// TIA Portal V18 export
DATA_BLOCK "Debug"   // DB5
{ S7_Optimized_Access := 'TRUE' }
VERSION : 0.1
// stored: AutoNumber false, DBAccessibleFromOPCUA true, DBAccessibleFromWebserver true, IsOnlyStoredInLoadMemory false, IsRetainMemResEnabled false, IsWriteProtectedInAS false, MemoryReserve 100
   VAR RETAIN
      SERVO_A1_LEGACY_MODE : Bool;
      SERVO_A2_LEGACY_MODE : Bool;
      SERVO_A3_LEGACY_MODE : Bool;
      SERVO_A4_LEGACY_MODE : Bool;
   END_VAR
BEGIN
END_DATA_BLOCK
